Staubli VAL3: safeCalibration.dtx

bool bEnded
bool bFinished
bool bResult
dio dIrefWarning = {link=Rsi9IO\IrefWarning}
dio dIsafePos = {link=Rsi9IO\IsafePos}
dio dIsafeRec = {link=Rsi9IO\IsafeRec}
dio dIsafeVel = {link=Rsi9IO\IsafeVel}
dio dIwaitingRestart = {link=Rsi9IO\IwaitingRestart}
dio dQrefPos1 = {link=Rsi9IO\QrefPos1}
dio dQrefPos2 = {link=Rsi9IO\QrefPos2}
dio dQresetRef = {link=Rsi9IO\QresetRef}
jointRx jInter[2]
  [0] = {j1=16.747153, j2=23.215229, j3=121.00356449, j4=36.67895, j5=59.788219, j6=-56.84014}
  [1] = {j1=15.334778, j2=29.352505, j3=112.42629, j4=211.510021, j5=-74.522323, j6=-55.937398}
jointRx jSafeReference1 = {j1=-15.981558, j2=6.260298, j3=120.160224, j4=31.4667, j5=66.893497, j6=-29.887624}
jointRx jSafeReference2 = {j1=-3.793248, j2=1.0269555, j3=124.00918551, j4=-180.851639, j5=-30.387886, j6=-41.572914}
jointRx jStart = {j1=-3.793236, j2=0.748011, j3=89.934189, j4=2.918087, j5=83.292851, j6=-41.834364}
jointRx jTmp
jointRx jTolerance = {j1=0.5, j2=0.5, j3=0.5, j4=0.5, j5=0.5, j6=0.5}
mdesc mNomSpeed
num nPrevSafeRefStatus
num nSafeRefStatus
pointRx pTmp = {fatherId=world[0]}
string sBtnFinished
string sHmiBgn{}
  [CurrentStatus] = {}
  [Processing] = {}
  [QrefPos1] = {}
  [QrefPos2] = {}
  [ReqAction] = {}
  [SafePosition] = {}
  [SafeRecovery] = {}
  [SafeVelocity] = {}
string sHmiColor{}
  [CurrentStatus] = {}
  [Processing] = {}
  [QrefPos1] = {}
  [QrefPos2] = {}
  [ReqAction] = {}
  [SafePosition] = {}
  [SafeRecovery] = {}
  [SafeVelocity] = {}
string sHmiColorDef{}
  [DefaultBgn] = {}
  [DefaultColor] = "black"
  [ErrorBgn] = "red"
  [ErrorColor] = "white"
  [InProgressBgn] = "green"
  [InProgressColor] = "black"
  [OffBgn] = "grey"
  [OffColor] = "white"
  [OkBgn] = "lime"
  [OkColor] = "black"
  [OnBgn] = "lime"
  [OnColor] = "black"
  [WarningBgn] = "orange"
  [WarningColor] = "black"
string sHmiStatusBgn{}
  [Checked] = {}
  [Defined] = {}
  [Invalid] = {}
  [Lost] = {}
  [Reset] = {}
  [Warning] = {}
string sHmiStatusColor{}
  [Checked] = {}
  [Defined] = {}
  [Invalid] = {}
  [Lost] = {}
  [Reset] = {}
  [Warning] = {}
string sHmiTxt{}
  [CurrentStatus] = {}
  [Processing] = {}
  [QrefPos1] = {}
  [QrefPos2] = {}
  [ReqAction] = {}
  [SafePosition] = {}
  [SafeRecovery] = {}
  [SafeVelocity] = {}
string sVersion
trsf trAppro
dio dQNoSafePos = {link=Rsi9IO\QnoSafePos}
dio dUSID1 = {link=Rsi9IO\IusiD1}
